{attribute addProperty BoxType "KL8548"}
{attribute addProperty Id "Channel_1Channel_B0A8062F00Channel_2Channel_B0A8062F00Channel_3Channel_B0A8062F00Channel_4Channel_B0A8062F00Channel_5Channel_B0A8062F00Channel_6Channel_B0A8062F00Channel_7Channel_B0A8062F00Channel_8Channel_B0A8062F00"}
{attribute addProperty CRC "2892660333"}
{attribute addProperty SizeInBites "0"}
{attribute addProperty SizeInBytes "0"}
TYPE KL8548_AC6A7E6D :
STRUCT
	{attribute addProperty Name "Channel_1"}
	Channel_1 : Channel_B0A8062F;
	{attribute addProperty Name "Channel_2"}
	Channel_2 : Channel_B0A8062F;
	{attribute addProperty Name "Channel_3"}
	Channel_3 : Channel_B0A8062F;
	{attribute addProperty Name "Channel_4"}
	Channel_4 : Channel_B0A8062F;
	{attribute addProperty Name "Channel_5"}
	Channel_5 : Channel_B0A8062F;
	{attribute addProperty Name "Channel_6"}
	Channel_6 : Channel_B0A8062F;
	{attribute addProperty Name "Channel_7"}
	Channel_7 : Channel_B0A8062F;
	{attribute addProperty Name "Channel_8"}
	Channel_8 : Channel_B0A8062F;
END_STRUCT
END_TYPE

(* stored: Version 1.2.0.0, ProductVersion 3.1.4024.9
   DUT KL8548_AC6A7E6D: Id {92c60ce8-58a4-47bf-b8c3-880c110e1fc0} *)
